(* CoDeSys 2.3.9.41 project: Котел_розжиг new.pro *)
(* Libraries: Standard.lib 4.10.05 11:14:46, SYSLIBCALLBACK.LIB 26.9.08 16:43:52, Util.lib 18.5.10 15:14:28, SysLibFile.lib 23.9.04 10:11:36 *)

(* Global variable list: Global_Variables *)
VAR_GLOBAL

	(*Ошибка *)
	Error:BOOL;
	codeError:WORD;
	errorMsg:STRING;
	errorCounter:INT;
	resetError:BOOL;
	errorArray: ARRAY[0..10 ] OF SensError;

	(*Тригеры*)
	stopTrig: F_TRIG;
	startTrig: F_TRIG;

	(* вода*)
	tempSpOut:REAL; (*Уставка*)
	waterRegulMech : waterRegulMech;



	(*flame*)
	igniter:BOOL;

	(*state*)
	start:BOOL;
	stop:BOOL;
	startBoiler:BOOL;
	gasMode:BOOL;
	oilMode:BOOL;
	isFlameStart:BOOL;
	flameStart:BOOL;

	(*Датчики *)
	gasConsum:REAL;
	oilConsum:REAL;
	waterInTemp:REAL;
	waterOutTemp:REAL;
	waterOutPressure:REAL;
	waterOutConsum:REAL;
	flameSensor:BOOL;
	conceCO2Sensor:REAL;
	oilPressureSensor:REAL;
	gasPressureSensor:REAL;

	(*Блок ошибок*)
	gasConsumError:SensError;
	oilConsumError:SensError;
	waterInTempError:SensError;
	waterOutTempError:SensError;
	waterOutPressureError:SensError;
	waterOutConsumError1:SensError;
	flameSensorError:SensError;
	conceCO2SensorError:SensError;
	oilPressureSensorError:SensError;
	gasPressureSensorError:SensError;
	fanFlameError:SensError;
	fanOutError:SensError;

	(*Клапана*)
	valveWaterTempIn:REAL;
	valveWaterTempOut:REAL;
	valveErrorOil:BOOL;
	valveErrorGas:BOOL;
	valveOilIn:BOOL;
	valveGasIn:BOOL;
	valveStartFlameOil:REAL;
	valveStartFlameGas:REAL;
	valveMainFlameOil:BOOL;
	valveMainFlameGas:BOOL;
	valveAeratorIn:BOOL;
	valveAeratorOut:BOOL;

	(*Вентиляторы*)
	fanFlame:REAL;
	fanOut:REAL;
	fanFlameBlock, fanOutBlock:fan;


	(*PID*)
	pidReg:myPid;
	spMinPidOut:WORD;
	spMaxPidOut:WORD;
	pidOffset, pidOffsetOld: WORD;

	(*Таймер*)
	saveParamTimer:TON;
	waterStartTON:TON;

	(*Util*)
	oilFlameMecanism:flameMecanism;
	gasFlameMecanism:flameMecanism;
	change: ARRAY[0..10 ] OF BOOL;

END_VAR

(* Data type *)
TYPE OptionsBoiler :
STRUCT
	gasMode:BOOL;
	oilMode:BOOL;
	start:BOOL;
	stop:BOOL;
END_STRUCT
END_TYPE

(* POU PLC_PRG, ST *)
PROGRAM PLC_PRG
VAR
	i: INT;
END_VAR
initParam;
stopStart;
sensControl;
airControl;
startFlameProcess;
waterControl;
errorHandle;
END_PROGRAM
ACTION airControl:
	fanFlameBlock(
	on:= start AND NOT Error,
	errorIn:= Error,
	gasMode:= gasMode,
	oilMode:= oilMode,
	valuePressureOil:= oilPressureSensor ,
	valuePressureGas:=gasPressureSensor,
	needPressureOil:= 300,(*0.. 100%  // - 50 .. 50 *)
	needPressureGas:= 23,(*0..100%  // - 50 .. 50 *)
	allowableError:=5,
	delayError:= t#10s,
	valueFanOut => fanFlame,
	errorOut =>(*В ошибку вентилятора*)
		);

	fanOutBlock(
	on:= start AND NOT Error,
	errorIn:= Error,
	gasMode:= TRUE ,(*Всегда один режим*)
	oilMode:= ,
	valuePressureOil:=  ,
	valuePressureGas:=  conceCO2Sensor,
	needPressureOil:= ,(*0.. 100%  // - 50 .. 50 *)
	needPressureGas:= 30,(*0..100%  // - 50 .. 50 *)
	allowableError:=15,
	delayError:= t#10s,
	valueFanOut => fanOut,
	errorOut =>(*В ошибку вентилятора*)
	);
END_ACTION
ACTION errorHandle:
errorCounter := BOOL_TO_INT( gasConsumError.errorOut) +
	BOOL_TO_INT(oilConsumError.errorOut) +
	BOOL_TO_INT(waterInTempError.errorOut) +
	BOOL_TO_INT(waterOutTempError.errorOut) +
	BOOL_TO_INT(waterOutPressureError.errorOut) +
	BOOL_TO_INT(waterOutConsumError1.errorOut) +
	BOOL_TO_INT(flameSensorError.errorOut) +
	BOOL_TO_INT(conceCO2SensorError.errorOut )+
	BOOL_TO_INT(oilPressureSensorError.errorOut)+
	BOOL_TO_INT(gasPressureSensorError.errorOut);


errorArray[0] :=gasConsumError;
errorArray[1] :=	oilConsumError;
errorArray[2] :=	waterInTempError;
errorArray[3] :=	waterOutTempError;
errorArray[4] :=	waterOutPressureError;
errorArray[5] :=	waterOutConsumError1;
errorArray[6] :=	flameSensorError;
errorArray[7] :=	conceCO2SensorError;
errorArray[8] :=	oilPressureSensorError;
errorArray[9] :=	gasPressureSensorError;

FOR i := 0 TO errorCounter - 1 DO
	errorMsg := CONCAT(errorMsg , '           ' );
	errorMsg := CONCAT(errorMsg , errorArray[i].errorMsgOut);
	i := i+1;
END_FOR;

errorMsg :=CONCAT( gasConsumError.errorMsgOut , oilConsumError.errorMsgOut) ;

Error :=( gasConsumError.errorOut OR
	oilConsumError.errorOut OR
	waterInTempError.errorOut OR
	waterOutTempError.errorOut OR
	waterOutPressureError.errorOut OR
	waterOutConsumError1.errorOut OR
	flameSensorError.errorOut OR
	conceCO2SensorError.errorOut OR
	oilPressureSensorError.errorOut OR
	gasPressureSensorError.errorOut ) AND NOT resetError ;
END_ACTION
ACTION initParam:
IF gasConsum = 0 AND NOT change[0]   THEN
	 gasConsum:=300;
	change[0]  := TRUE;
 END_IF
(*_______________________________________________________________*)

IF oilConsum = 0 AND NOT change[1]  THEN
	 oilConsum:=300;
	change[1]  := TRUE;
 END_IF
(*_______________________________________________________________*)

IF waterInTemp = 0 AND NOT change[2]   THEN
	waterInTemp:=50;
	change[2] := TRUE;
 END_IF
(*_______________________________________________________________*)
IF waterOutTemp = 0 AND NOT change[3]   THEN
	waterOutTemp:=150;
	change[3]  := TRUE;
 END_IF
(*_______________________________________________________________*)
IF waterOutPressure = 0 AND NOT change[4]   THEN
	waterOutPressure:=5;
	change[4]  := TRUE;
 END_IF
(*_______________________________________________________________*)
IF waterOutConsum = 0 AND NOT change[5]   THEN
	waterOutConsum:=5;
	change[5]  := TRUE;
 END_IF


(*_______________________________________________________________*)
IF conceCO2Sensor = 0 AND NOT change[6]  THEN
	conceCO2Sensor:=50;
	change[6] := TRUE;
 END_IF
(*_______________________________________________________________*)
IF gasPressureSensor = 0 AND NOT change[7]  THEN
	gasPressureSensor:=23;
	change[7] := TRUE;
 END_IF
(*_______________________________________________________________*)
IF oilPressureSensor = 0 AND NOT change[8]  THEN
	oilPressureSensor:=300;
	change[8] := TRUE;
 END_IF

IF tempSpOut = 0 AND NOT change[9]  THEN
	tempSpOut := 150;
	change[9] := TRUE;
 END_IF
END_ACTION
ACTION sensControl:
	gasConsumError(
	on:=gasMode,
	errorMsg:= 'Ошибка датчика расхода газа',
	value := gasConsum  ,
	errorValueMax:=400,
	errorValueMin:=200,
	errorOut => codeError.7
	);
(*_______________________________________________________________*)
	oilConsumError(
	on:=oilMode,
	errorMsg:= 'Ошибка датчика расхода мазута',
	value := oilConsum  ,
	errorValueMax:=400,
	errorValueMin:=200,
	errorOut => codeError.0
	);
(*_______________________________________________________________*)
	waterInTempError(
	on:=start,
	errorMsg:= 'Ошибка датчика температуры воды на входе',
	value := waterInTemp ,
	errorValueMax:=65,
	errorValueMin:=40,
	errorOut => codeError.1
	);
(*_______________________________________________________________*)
	waterOutTempError(
	on:=start,
	errorMsg:= 'Ошибка датчика температуры воды на выходе',
	value :=waterOutTemp  ,
	errorValueMax:=160,
	errorValueMin:=140,
	delay:= t#120s,
	errorOut => codeError.2
	);
(*_______________________________________________________________*)
	waterOutPressureError(
	on:=start,
	errorMsg:= 'Ошибка датчика давления воды на выходе',
	value :=  waterOutPressure,
	errorValueMax:=0,
	errorValueMin:=10,
	delay:= t#120s,
	errorOut => codeError.3
	);
(*_______________________________________________________________*)
	waterOutConsumError1(
	on:=start,
	errorMsg:= 'Ошибка датчика расхода воды на выходе',
	value :=  waterOutConsum,
	errorValueMax:=0,
	errorValueMin:=10,
	delay:= t#120s,
	errorOut => codeError.4
	);
(*_______________________________________________________________*)

	flameSensorError(
	on:=start,
	justError:= oilFlameMecanism.flameProcessErrorFlag1
				OR gasFlameMecanism.flameProcessErrorFlag1,
	errorMsg:= 'Ошибка розжига котла',
	oneErrorMode:=TRUE,
	delay:= t#5s,
	errorOut => codeError.5
	);


(*_______________________________________________________________*)
	conceCO2SensorError(
	on:=start,
	errorMsg:= 'Ошибка датчика концентрации уходящих газов',
	value :=  conceCO2Sensor,
	errorValueMax:=100,
	errorValueMin:=0,
	errorOut => codeError.6
	);
(*_______________________________________________________________*)

	gasPressureSensorError(
	on:=gasMode,
	errorMsg:= 'Ошибка датчика давления газа',
	value := gasPressureSensor  ,
	delay:= t#30s,
	errorValueMax:=25,
	errorValueMin:=20,
	errorOut => codeError.7
	);
(*_______________________________________________________________*)

	oilPressureSensorError(
	on:=oilMode,
	errorMsg:= 'Ошибка датчика давления мазута',
	value := oilPressureSensor  ,
	delay:= t#30s,
	errorValueMax:=400,
	errorValueMin:=170,
	errorOut => codeError.0
	);

	fanOutError(
	on:=start,
	justError:= fanOutBlock.errorOut,
	errorMsg:= 'Ошибка розжига котла',
	oneErrorMode:=TRUE,
	delay:= t#30s,
	errorOut => codeError.5
	);

	fanFlameError(
	on:=start,
	justError:=  fanFlameBlock.errorOut,
	errorMsg:= 'Ошибка розжига котла',
	oneErrorMode:=TRUE,
	delay:= t#30s,
	errorOut => codeError.5
	);
END_ACTION
ACTION startFlameProcess:
flameSensor:= flameStart AND start;


igniter := oilFlameMecanism.igniterLocal OR gasFlameMecanism.igniterLocal;

gasFlameMecanism(
	on:= gasMode AND (NOT Error) AND NOT oilMode,
	igniterTryCounter:= 10,
	valveError => valveErrorGas,
	valveIn =>valveGasIn,
	valveStartFlame =>valveStartFlameGas,
	valveMain => valveMainFlameGas,
	igniterLocal => ,
	flameProcessErrorFlag1 => );

oilFlameMecanism(
	on:= oilMode AND (NOT Error) AND NOT gasMode,
	igniterTryCounter:= 10,
	valveError => valveErrorOil,
	valveIn =>valveOilIn,
	valveStartFlame =>valveStartFlameOil,
	valveMain => valveMainFlameOil,
	igniterLocal => ,
	flameProcessErrorFlag1 => );
END_ACTION
ACTION stopStart:
IF startBoiler THEN
	start:=TRUE;
	stop:=FALSE;
 ELSE stop:=TRUE;
	start:=FALSE;
 END_IF

IF Error THEN
	 stop:=TRUE;
	start:=FALSE;
END_IF
IF oilMode THEN gasMode := FALSE; oilMode := TRUE; ELSE gasMode := TRUE; oilMode := FALSE;  END_IF
IF gasMode THEN gasMode := TRUE; oilMode := FALSE; ELSE  gasMode := FALSE; oilMode := TRUE;  END_IF
END_ACTION
ACTION waterControl:
waterStartTON(IN:=flameSensor AND start AND NOT error , PT:= t#30s);

valveWaterTempIn := SEL(NOT(waterStartTON.ET = T#0s ) , 0, 100);
valveAeratorIn:= NOT(waterStartTON.ET = T#0s ) OR waterStartTon.Q;
valveAeratorOut:= NOT(waterStartTON.ET = T#0s ) OR waterStartTon.Q;

waterRegulMech(
	on:= waterStartTon.Q	AND
		waterInTempError.resultsIsRight AND
		waterOutPressureError.resultsIsRight AND
		 waterOutConsumError1.resultsIsRight ,
	error:=Error,
	value:= waterOutTemp,
	needValue:=tempSpOut ,(*150*)
	allowableError:= 10,
	delayError:= t#2m,
	 valueWaterOut => valveWaterTempOut ,
	errorOut =>
	);

(*
IF NOT Error AND NOT stop AND  NOT(waterStartTON.ET = T#0s )    THEN

	IF spMinPidOut>=spMaxPidOut THEN spMaxPidOut:=spMinPidOut+1; END_IF

	IF PidReg.Y<=spMinPidOut THEN
		pidOffset:=spMinPidOut;
		ELSIF PidReg.Y>=spMaxPidOut THEN
			pidOffset:=spMaxPidOut;
			ELSE
				pidOffset:=pidOffsetOld;
	END_IF
	PidReg(
		actual:=waterOutTemp,
		sp:=tempSpOut,
		spShift:=4,
		KP:=10/100,(*Чисто рандом*)
		TN:=10,(*да*)
		TV:=,
		yManual:=0,
		yOffset:=pidOffset,
		yMin:=50,
		yMax:=165,
		manual:= TRUE,(*pid mode*)
		deadZone:=0.25,
		reset:=PidReg.overflow OR  Error AND  stop AND  waterStartTON.ET = T#0s  ,
		(*Выхода*)
		Y=>);

END_IF;
*)
END_ACTION

(* POU saveLoadParamFile, ST *)
PROGRAM saveLoadParamFile
VAR
	file:				DWORD;
	optBoiler:			OptionsBoiler;

	optionSaveFT: F_TRIG;
	loadTON: TON;
	optionsLoadFT: F_TRIG;
	startLoad: BOOL:=TRUE;
END_VAR
loadTON(IN:=startLoad, PT:=T#50ms);
IF loadTON.Q THEN startLoad:=FALSE; END_IF

optionsLoadFT(CLK:= startLoad);


saveParamTimer(IN:= NOT saveParamTimer.Q , PT:=T#10s);

optionSaveFT(CLK:=saveParamTimer.Q);

IF optionSaveFT.Q THEN
	optBoiler.gasMode := gasMode;
	optBoiler.oilMode := oilMode;
	optBoiler.start := start;
	optBoiler.stop := stop;

	file:=SysFileOpen('options', 'w');
	SysFileWrite(file, ADR(optBoiler), SIZEOF(optBoiler));
	SysFileClose(file);
END_IF

IF optionsLoadFT.Q THEN
	file:=SysFileOpen('options', 'r');
	SysFileRead(file, ADR(optBoiler), SIZEOF(optBoiler));
	SysFileClose(file);

	gasMode:= optBoiler.gasMode;
	oilMode:= optBoiler.oilMode;
	start:=optBoiler.start ;
	stop := optBoiler.stop;
END_IF
END_PROGRAM

(* POU lib/Blinker, ST *)
FUNCTION_BLOCK Blinker
(* Function block to simulate a turn signal *)
VAR_INPUT
	enable:		BOOL;	(* TRUE:run Blink, FALSE: OUT keeps its value*)
	timeLow:	TIME;	(* Time for OUT=FALSE *)
	timeHigh:	TIME;	(* Time for OUT=TRUE *)
END_VAR
VAR_OUTPUT
	out:		BOOL;	(* output variable, starting with FALSE *)
END_VAR
VAR
	clock:		TP;
END_VAR
clock;								(* call Timer *)
IF clock.Q=FALSE AND enable THEN	(* time passed or init *)
	clock(IN:=FALSE);				(* reset Timer *)
	clock(IN:=TRUE);				(* restart Timer *)
	IF Out=FALSE THEN
		clock.PT:=timeHigh;
	ELSE
		clock.PT:=timeLow;
	END_IF;
	out := NOT out;					(* invert *)
END_IF

IF NOT enable THEN Out:=FALSE; END_IF
END_FUNCTION_BLOCK

(* POU lib/Deriv, ST *)
(* function block to approximate the derivative of a value *)
(* to calculate this, always four values are used in order to be as exact as possible *)
FUNCTION_BLOCK Deriv
VAR_INPUT
	in:REAL;		(* input variable *)
	tm:DWORD;		(* time since last call in msec *)
	reset:BOOL;		(* reset: set OUT to zero *)
END_VAR
VAR_OUTPUT
	out:REAL;		(* derivative *)
END_VAR
VAR
	X3,X2,X1:REAL;
	T2,T1:DWORD;
	init:BOOL:=TRUE;
END_VAR
IF init OR reset THEN
	X1:=in;
	X2:=in;
	X3:=in;
	out:=0;
	init:=FALSE;
ELSE
	IF tm>0 THEN
		out:=(3*(in-X3)+X1-X2)/((3*T2+4*T1+3*tm))*1000;
		X3:=X2;
		X2:=X1;
		X1:=in;
		T2:=T1;
		T1:=tm;
	END_IF;
END_IF;
END_FUNCTION_BLOCK

(* POU mech/fan, ST *)
FUNCTION_BLOCK fan
VAR_INPUT
	on:BOOL;
	errorIn:BOOL;
	gasMode:BOOL;
	oilMode:BOOL;
	valuePressureOil:REAL;
	valuePressureGas:REAL;
	needPressureOil:REAL;
	needPressureGas:REAL;
	allowableError:REAL;
	delayError:TIME;
END_VAR
VAR_OUTPUT
	 valueFanOut:REAL;
	errorOut:BOOL;
END_VAR
VAR
	realErrorTimer:TON;
	makeFixSpeed:BOOL;
	valuePressure:REAL;
	needPressure:REAL;
	errorTimer:TON;
	plusValueBlinker:BLINK;
	plusValueTrig: R_TRIG;
	minusValueBlinker: BLINK;
	minusValueTrig: R_TRIG;
END_VAR
IF gasMode THEN
	valuePressure:= valuePressureGas;
	needPressure := needPressureGas;
END_IF

IF oilMode THEN
	valuePressure:= valuePressureOil;
	needPressure := needPressureOil;

END_IF

IF errorIn THEN
	valueFanOut:= 100;
	realErrorTimer(In:=TRUE, PT:= delayError);
	IF realErrorTimer.Q THEN
		valueFanOut:= 0;
	END_IF
  END_IF

IF valueFanOut< 0 THEN
	valueFanOut:= 0;
END_IF
IF valueFanOut > 100 THEN
	valueFanOut:= 100;
END_IF

IF on THEN
	IF valuePressure > needPressure + allowableError OR valuePressure < needPressure - allowableError THEN
		errorTimer(In:=TRUE, PT:= delayError);
		IF errorTimer.Q THEN
			errorOut:=TRUE;
		END_IF

	ELSE
		errorTimer(In:=FALSE, PT:= delayError);
		errorOut:=FALSE;
	END_IF
	IF valuePressure > needPressure + allowableError  AND NOT makeFixSpeed THEN
		plusValueBlinker(enable:=TRUE,
				timeLow:= t#500ms,
				timeHigh:=t#500ms );
		plusValueTrig(CLK:= plusValueBlinker.out);

		IF plusValueTrig.Q  THEN  valueFanOut := valueFanOut - 1; END_IF

	END_IF
	IF valuePressure <  needPressure - allowableError AND NOT makeFixSpeed  THEN
		minusValueBlinker(enable:=TRUE,
				timeLow:= t#500ms,
				timeHigh:=t#500ms );
		minusValueTrig(CLK:= minusValueBlinker.out);

		IF minusValueTrig.Q  THEN  valueFanOut := valueFanOut + 1; END_IF

	END_IF
	makeFixSpeed:= valuePressure < needPressure + allowableError AND valuePressure > needPressure - allowableError ;
END_IF
END_FUNCTION_BLOCK

(* POU mech/flameMecanism, ST *)
FUNCTION_BLOCK flameMecanism
VAR_INPUT
	on:BOOL;
	igniterTryCounter:INT;

END_VAR
VAR_OUTPUT
	valveError:BOOL;
	valveIn:BOOL;
	valveStartFlame:REAL;
	valveMain:BOOL;
	igniterLocal:BOOL;
	stopFlag:BOOL;
	startFlag:BOOL;
	flameProcessErrorFlag1 :BOOL;


END_VAR
VAR
	igniterTryCounterLocal:INT;
	flameStartCounter:INT;
	valveStartFlameMech:valveStartFlameMech;
	flameStartBlinker:BLINK;
	flameStartTrig:R_TRIG;
END_VAR
igniterTryCounterLocal:= igniterTryCounter - 1;
IF on AND start AND NOT stop THEN
	IF flameStartCounter= 0 THEN
		flameProcessErrorFlag1 :=FALSE;
		valveError:=TRUE;
		valveIn:=TRUE;
		startFlag:=TRUE;
		stopFlag:=FALSE;
	END_IF
	flameStartBlinker(enable:= start AND NOT flameSensor,
						timeLow:= t#1s,
						timeHigh:= t#1s);
	flameStartTrig(CLK:= flameStartBlinker.out);

	igniterLocal:=  flameStartBlinker.out;

	(*flame NOT START  check 3 times*)
	IF flameStartCounter <=  igniterTryCounterLocal - 1 AND flameStartTrig.Q AND igniterLocal THEN
		flameStartCounter := flameStartCounter + 1;

	END_IF
	IF flameStartCounter = igniterTryCounterLocal THEN
		stopFlag:=TRUE;
		startFlag:=FALSE;
		flameProcessErrorFlag1 :=TRUE;
		valveError:=FALSE;
		valveIn:=FALSE;
		valveStartFlame:= 0;
		igniterLocal:=FALSE;
	END_IF

	(*flame START*)
	IF flameSensor THEN
		isFlameStart:= TRUE;
		igniterLocal:=FALSE;
	END_IF

	valveStartFlameMech(isStart:= startFlag,
			isStop:=flameSensor,
			valveCurrentPercent:= valveStartFlame ,
		valvePercent =>valveStartFlame ,
		valveMain => valveMain);

END_IF

IF stop  OR flameProcessErrorFlag1 THEN
	startFlag:=FALSE;
	valveError:=FALSE;
	valveIn:=FALSE;
	valveMain:=FALSE;
	valveStartFlame:= 0;
	igniterLocal:=FALSE;
END_IF
END_FUNCTION_BLOCK

(* POU mech/valveStartFlameMech, ST *)
FUNCTION_BLOCK valveStartFlameMech
VAR_INPUT
	isStart:BOOL;
	isStop:BOOL;
	valveCurrentPercent:REAL;
END_VAR
VAR_OUTPUT
	valvePercent:REAL;
	valveMain:BOOL;
END_VAR
VAR

	flameStartBlinker:BLINK;
	flameStartTrig:R_TRIG;

	flameBeginBlinker:BLINK;
	flameBeginTrig:R_TRIG;
END_VAR
IF valvePercent = 0 THEN valvePercent:= valveCurrentPercent; END_IF

IF isStart THEN
		flameStartBlinker(enable:= start AND NOT flameSensor,
							timeLow:= t#500ms,
							timeHigh:= t#500ms);

		flameStartTrig(CLK:= flameStartBlinker.out);

		IF	 flameStartTrig.Q  AND (NOT isStop)THEN
			valvePercent:= valvePercent + 3;
		END_IF
END_IF

IF isStop THEN
			valvePercent:= 0;
			valveMain:=TRUE;

END_IF
END_FUNCTION_BLOCK

(* POU lib/Integ, ST *)
(* function block to approximate the integral of IN over the time *)
FUNCTION_BLOCK Integ
VAR_INPUT
	in:REAL;				(* input variable *)
	tm:DWORD;				(* time since last call in msec *)
	reset:BOOL;				(* reset: OUT is set to zero and OVERFLOW to false *)
END_VAR
VAR_OUTPUT
	out:REAL;				(* value of the integral *)
	overflow:BOOL:=FALSE;	(* overflow *)
END_VAR
VAR
END_VAR
IF reset THEN
	out:=0;
	overflow:=FALSE;
ELSIF NOT overflow  THEN
	IF 1E38 - in*tm < out OR -1E38 - in*tm > out THEN
		overflow:=TRUE;
	ELSE
		out:=out+in*tm/1000;
	END_IF;
END_IF;
END_FUNCTION_BLOCK

(* POU lib/myPid, ST *)
FUNCTION_BLOCK myPid
VAR_INPUT
	actual:		REAL;	(*Текущее значение*)
	sp:			REAL;	(*Уставка*)
	spShift:	REAL;	(*Сдвиг уставки для уменьшения скорости ПИД на большом диапазоне, если SPShift<DeadZone то выкл*)
	KP:			REAL;	(*Пропорциональный коэффициент*)
	TN:			REAL;	(*Интегральный коэффициент*)
	TV:			REAL;	(*Время интегрирования в *)
	yManual:	REAL;	(*Y равен этому значению когда MANUAL=TRUE*)
	yOffset:	REAL;	(*Смещение выхода на старте*)
	yMin:		REAL;	(*Минимум выхода*)
	yMax:		REAL;	(*Максимум выхода*)
	manual:		BOOL;	(*Y=YManual когда MANUAL=TRUE *)
	reset:		BOOL;	(*Сброс регулятора Y=YOffset*)
	deadZone:	REAL;	(*Ширина зоны нечувствительности*)
END_VAR
VAR_OUTPUT
	Y:				REAL;			(*Выходное значение*)
	limitsActive:	BOOL:=FALSE;	(*Достигнуты лимиты выхода YMin, YMax *)
	overflow:		BOOL:=FALSE;	(*Переполнение интегральной части*)
END_VAR
VAR
	clock:			TON;
	I: 				Integ;
	D: 				Deriv;
	tmDiff: 		DWORD;
	error: 			REAL;
	init: 			BOOL:=TRUE;
END_VAR
IF TN>0 AND KP<> 0 AND (NOT overflow OR reset OR manual) THEN
	sp:=SEL(spShift>DeadZone, sp, SEL(sp-spShift>actual, sp, actual+spShift));
	error := SEL( ABS(sp-actual)<deadZone, sp-actual, 0);			(* Regeldifferenz *)

	IF reset OR init OR manual THEN	(* Reset oder Handbetrieb *)
		I(Reset:=TRUE);
		D(Reset:=TRUE);
		overflow:=FALSE;
		limitsActive:=FALSE;
		IF reset OR init THEN
			Y := yOffset;
			init:=FALSE;
			ELSIF manual THEN
				Y := yManual;
		END_IF
		tmDiff:=0;
		clock(IN:=FALSE);									(* Timer neu starten *)
		clock(PT:=t#1h, IN:=TRUE);
		ELSE
			clock;											(* Timer abfragen *)
			tmDiff:=TIME_TO_DWORD(Clock.ET);				(* Zeitdifferenz seit letztem Aufruf *)
	END_IF;

	IF tmDiff>0 THEN
		clock(IN:=FALSE);									(* Timer neu starten *)
		clock(PT:=t#1h, IN:=TRUE);

		D(IN:=error, TM:=tmDiff, reset:=FALSE);				(* Differential abschätzen *)
		I(IN:=error, TM:=SEL(limitsActive, tmDiff, 0), reset:=FALSE);				(* Integral abschätzen *)

		overflow := I.overflow;
		IF NOT overflow THEN
			Y:=yOffset+KP*(error+I.out/TN+D.out*TV);
			IF Y>1E30 OR Y<-1E30 THEN					(* Overflow steht bevor, darf aber eigentlich nicht passieren *)
				overflow:=TRUE;
			END_IF;

			limitsActive:=FALSE;
			IF yMax>yMin AND Y>=yMax  THEN				(* Stellwert-Obergrenze ьberschritten *)
				limitsActive:=TRUE;
				IF KP<>0 THEN
					I(IN:=(yMax-Y)*TN/KP, TM:=1000, Reset:=FALSE);	(* Integral korrigieren *)
				END_IF
				Y:=yMax;
			END_IF;

			IF yMax>yMin AND Y<=yMin THEN					(* Stellwert-Untergrenze unterschritten *)
				limitsActive:=TRUE;
				IF KP<>0 THEN
					I(IN:=(yMin-Y)*TN/KP, TM:=1000, Reset:=FALSE);	(* Integral korrigieren *)
				END_IF
				Y:=yMin;
			END_IF;
		END_IF;
	END_IF;

END_IF;
END_FUNCTION_BLOCK

(* POU mech/SensError, ST *)
FUNCTION_BLOCK SensError
VAR_INPUT
	value:REAL;
	on:BOOL;
	errorReset:BOOL;
	errorMsg:STRING;
	oneErrorMode:BOOL;
	justError:BOOL;
	errorValueMax:REAL;
	errorValueMin:REAL;
	delay:TIME:=t#10s;
END_VAR
VAR_OUTPUT
	errorOut:BOOL;
	resultsIsRight:BOOL;
	errorMsgOut:STRING;
END_VAR
VAR
	errorHandleTon: TON;
END_VAR
IF oneErrorMode THEN
	 errorValueMax := 1 ;
	errorValueMin:= -1;
 END_IF

IF ((value >= errorValueMax OR value <= errorValueMin) OR justError ) AND NOT resetError AND on THEN
	errorHandleTon(IN:= start AND NOT stop, PT:= delay);
	errorHandleTon;
	IF errorHandleTon.Q THEN
		 errorOut := TRUE;
		errorMsgOut:= errorMsg;
	END_IF
	ELSE
	errorMsgOut:= '';
 END_IF

resultsIsRight := (NOT errorOut) AND start AND on;
END_FUNCTION_BLOCK

(* POU mech/waterRegulMech, ST *)
FUNCTION_BLOCK waterRegulMech
VAR_INPUT
	on:BOOL;
	error:BOOL;
	value:REAL;
	needValue:REAL;(*150*)
	allowableError:REAL;
	delayError:TIME;
END_VAR
VAR_OUTPUT
	 valueWaterOut:REAL;
	errorOut:BOOL;
END_VAR
VAR
	errorTimer:TON;
	plusValueBlinker:BLINK;
	plusValueTrig: R_TRIG;
	minusValueBlinker: BLINK;
	minusValueTrig: R_TRIG;
END_VAR
IF on AND NOT error THEN
	IF value > needValue + allowableError AND value < needValue + allowableError THEN
		errorTimer(In:=TRUE, PT:= delayError);
		IF errorTimer.Q THEN
			errorOut:=TRUE;
		END_IF

	ELSE
		errorTimer(In:=FALSE, PT:= delayError);
		errorOut:=FALSE;
	END_IF
	IF value > needValue + allowableError  THEN
		plusValueBlinker(enable:=TRUE,
				timeLow:= t#500ms,
				timeHigh:=t#500ms );
		plusValueTrig(CLK:= plusValueBlinker.out);

		IF plusValueTrig.Q  THEN  valueWaterOut := valueWaterOut - 1; END_IF

	END_IF
	IF value <  needValue - allowableError  THEN
		minusValueBlinker(enable:=TRUE,
				timeLow:= t#500ms,
				timeHigh:=t#500ms );
		minusValueTrig(CLK:= minusValueBlinker.out);

		IF minusValueTrig.Q  THEN  valueWaterOut := valueWaterOut + 1; END_IF

	END_IF
END_IF
END_FUNCTION_BLOCK

(* Visualisation ignition
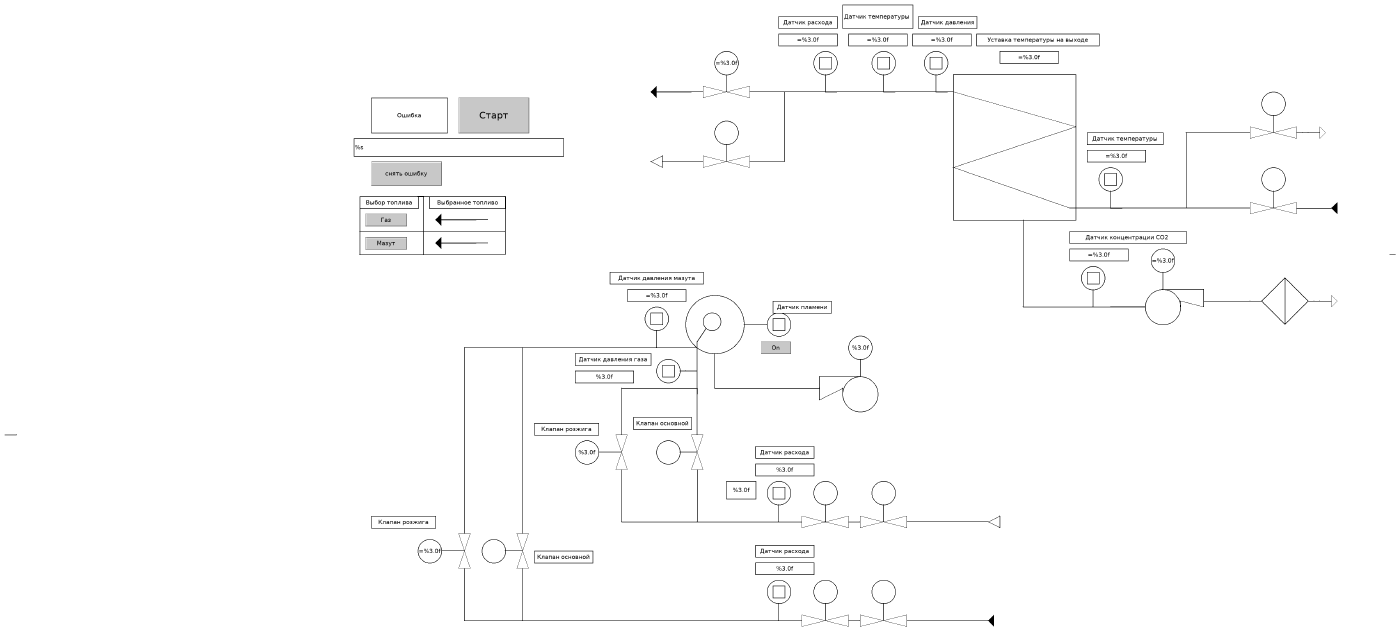
ellipse at (420,740)-(461,781): alarm colour if .valveMainFlameGas
ellipse at (280,740)-(321,781): text "%3.0f"; shows .valveStartFlameGas; alarm colour if .valveStartFlameGas; editable 0..100
ellipse at (610,810)-(651,851): alarm colour if .gasConsumError.resultsIsRight
ellipse at (500,520)-(531,551): alarm colour if .igniter
ellipse at (610,520)-(651,561): alarm colour if .flameSensor
ellipse at (790,810)-(831,851): alarm colour if .valveGasIn
rectangle at (590,750)-(691,771): text "Датчик расхода"
rectangle at (210,710)-(321,731): text "Клапан розжига"
rectangle at (380,700)-(481,721): text "Клапан основной"
button at (80,150)-(201,211): text "Старт"; toggles startBoiler
ellipse at (750,560)-(791,601): text "%3.0f"; shows .fanFlame; alarm colour if .fanFlame
button at (600,570)-(651,591): text "On"; toggles .flameStart
rectangle at (590,780)-(691,801): text "%3.0f"; shows .gasConsum; editable 0..1000
rectangle at (540,810)-(591,841): text "%3.0f"; shows PLC_PRG.consFuelSensor; editable 0..1000
ellipse at (690,810)-(731,851): alarm colour if .valveErrorGas
ellipse at (1460,270)-(1501,311): alarm colour if .valveWaterTempIn
ellipse at (690,70)-(731,111): shows .waterOutConsumError1.resultsIsRight
rectangle at (630,10)-(731,31): text "Датчик расхода"
rectangle at (630,40)-(731,61): text "=%3.0f"; shows .waterOutConsum; editable 0..1000
ellipse at (1270,410)-(1311,451): text "=%3.0f"; shows .fanOut; alarm colour if .fanOut
ellipse at (610,980)-(651,1021): alarm colour if .oilConsumError.resultsIsRight
ellipse at (790,980)-(831,1021): alarm colour if .valveOilIn
rectangle at (590,920)-(691,941): text "Датчик расхода"
rectangle at (590,950)-(691,971): text "%3.0f"; shows .oilConsum; editable 0..1000
ellipse at (690,980)-(731,1021): alarm colour if .valveErrorOil
ellipse at (120,910)-(161,951): alarm colour if .valveMainFlameOil
ellipse at (10,910)-(51,951): text "=%3.0f"; shows .valveStartFlameOil; alarm colour if .valveStartFlameOil; editable 0..100
rectangle at (-70,870)-(41,891): text "Клапан розжига"
rectangle at (210,930)-(311,951): text "Клапан основной"
ellipse at (520,190)-(561,231): alarm colour if .valveAeratorOut
ellipse at (1460,140)-(1501,181): alarm colour if .valveAeratorIn
ellipse at (790,70)-(831,111): alarm colour if .waterOutTempError.resultsIsRight
rectangle at (740,-10)-(861,31): text "Датчик температуры"
rectangle at (750,40)-(851,61): text "=%3.0f"; shows .waterOutTemp; editable 0..1000
ellipse at (880,70)-(921,111): alarm colour if .waterOutPressureError.resultsIsRight
rectangle at (870,10)-(971,31): text "Датчик давления"
rectangle at (860,40)-(961,61): text "=%3.0f"; shows .waterOutPressure; editable 0..1000
ellipse at (1180,270)-(1221,311): alarm colour if .waterInTempError.resultsIsRight
rectangle at (1160,210)-(1291,231): text "Датчик температуры"
rectangle at (1160,240)-(1261,261): text "=%3.0f"; shows .waterInTemp; editable 0..1000
ellipse at (1150,440)-(1191,481): alarm colour if .conceCO2SensorError.resultsIsRight
rectangle at (1130,380)-(1331,401): text "Датчик концентрации CO2"
rectangle at (1130,410)-(1231,431): text "=%3.0f"; shows .conceCO2Sensor; editable 0..100
button at (-80,350)-(-9,371): text "Газ"; toggles .gasMode
button at (-80,390)-(-9,411): text "Мазут"; toggles .oilMode
rectangle at (620,500)-(721,521): text "Датчик пламени"
rectangle at (620,500)-(721,521): text "Датчик пламени"
rectangle at (-90,320)-(11,341): text "Выбор топлива"
rectangle at (30,320)-(161,341): text "Выбранное топливо"
rectangle at (-70,150)-(61,211): text "Ошибка"; alarm colour if Error
ellipse at (400,510)-(441,551): alarm colour if .oilPressureSensorError.resultsIsRight
rectangle at (340,450)-(501,471): text "Датчик давления мазута"
rectangle at (370,480)-(471,501): text "=%3.0f"; shows .oilPressureSensor; editable 0..1000
ellipse at (420,600)-(461,641): alarm colour if .gasPressureSensorError.resultsIsRight
rectangle at (280,590)-(411,611): text "Датчик давления газа"
rectangle at (280,620)-(381,641): text "%3.0f"; shows .gasPressureSensor; editable 0..1000
rectangle at (-100,220)-(261,251): text "%s"; shows errorMsg
button at (-70,260)-(51,301): text "снять ошибку"; taps resetError
rectangle at (700,80)-(721,101): alarm colour if .waterOutConsumError1.errorOut
rectangle at (800,80)-(821,101): alarm colour if .waterOutTempError.errorOut
rectangle at (890,80)-(911,101): alarm colour if .waterOutPressureError.errorOut
rectangle at (1190,280)-(1211,301): alarm colour if .waterInTempError.errorOut
rectangle at (1160,450)-(1181,471): alarm colour if .conceCO2SensorError.errorOut
rectangle at (620,820)-(641,841): alarm colour if .gasConsumError.errorOut
rectangle at (430,610)-(451,631): alarm colour if .gasPressureSensorError.errorOut
rectangle at (410,520)-(431,541): alarm colour if .oilPressureSensorError.errorOut
rectangle at (620,990)-(641,1011): alarm colour if .oilConsumError.errorOut
rectangle at (620,530)-(641,551): alarm colour if .flameSensorError.errorOut
rectangle at (970,40)-(1181,61): text "Уставка температуры на выходе"
rectangle at (1010,70)-(1111,91): text "=%3.0f"; shows .tempSpOut; editable 0..1000
ellipse at (520,70)-(561,111): text "=%3.0f"; shows .valveWaterTempOut; alarm colour if .valveWaterTempOut
81 more shapes without text or variables
*)
